// TIA Portal V19 export
FUNCTION_BLOCK "CallEquipmentMotionCycle"   // FB150, LAD
AUTHOR : Siemens_FA_SUP
// stored: IsIECCheckEnabled true, MemoryReserve 100, Namespace Unit.Em2, SetENOAutomatically true
   VAR_OUTPUT
      error { ExternalAccessible := 'False'; ExternalVisible := 'False'; ExternalWritable := 'False'} : Bool;
   END_VAR
   VAR_IN_OUT
      syncNode : "Unit.Em2.typeSyncNode";
   END_VAR
BEGIN

REGION Network 1: Call Sequence
   // Add logic here, that should be executed in the Motion cycle. This logic called in OB MC_PreInterpolator. This could be e.g. immediate positioning commands.
END_REGION
END_FUNCTION_BLOCK
